{attribute 'GeneratedUsingTerminal: EPP1342-0001-0016'}
{attribute addProperty BoxType "EPP1342-0001-0016"}
{attribute addProperty Id "A_0024_EPP1342_0001_0017A_0024_EPP1342_0001_0017_FC9F5325378"}
{attribute addProperty CRC "2183154156"}
{attribute addProperty Size "378"}
TYPE A_0023_EPP1342_0001_0016_822049EC EXTENDS EPP1342_1FC0878B :
STRUCT
	{attribute addProperty Name "A_0024_EPP1342_0001_0017"}
	{attribute addProperty PreviousPort "A_0023(EPP1342-0001-0016) : D"}
	A_0024_EPP1342_0001_0017 : A_0024_EPP1342_0001_0017_FC9F5325;
END_STRUCT
END_TYPE

(* stored: Version 1.2.0.0, ProductVersion 3.1.4024.9
   DUT A_0023_EPP1342_0001_0016_822049EC: Id {f72cd63f-9ea1-4d2c-91aa-0c964918b43c} *)
